(* Logix 5000 project; controller Oki_4_23 vendor 1 type 14 code 77 rev 20.12; software revision 20.01 *)

TASK MainTask (continuous, watchdog 500 ms) : MainProgram

MODULES
   Controller : vendor 1 type 14 code 77 (CompactLogixL32EController 0, rev 20.12)
      LocalENB : 1769-L32E Ethernet Port (CompactLogixL32Ethernet 1, rev 20.11)
      Local : CompactBus (CompactVirtualAdapter 3, rev 20.11)
         INPUT_1 : 1769-IQ16 (Compact 1, rev 1.1, Input RPI 20 ms)
         OUTPUT : 1769-OB16 (Compact 2, rev 2.1, Output RPI 20 ms)
END_MODULES

VAR_GLOBAL   (* controller tags *)
   GREEN : ALIAS FOR Local:2:O.Data.13;
   RED : ALIAS FOR Local:2:O.Data.15;
   START1 : ALIAS FOR Local:1:I.Data.1;
   START2 : ALIAS FOR Local:1:I.Data.2;
   START3 : ALIAS FOR Local:1:I.Data.3;
   START4 : ALIAS FOR Local:1:I.Data.4;
   STOP : ALIAS FOR Local:1:I.Data.5;
   TIMER1 : TIMER := (PRE := 5000);
   TIMER2 : TIMER := (PRE := 5000);
END_VAR

PROGRAM MainProgram   (* main routine MainRoutine *)

ROUTINE MainRoutine   (* ladder *)
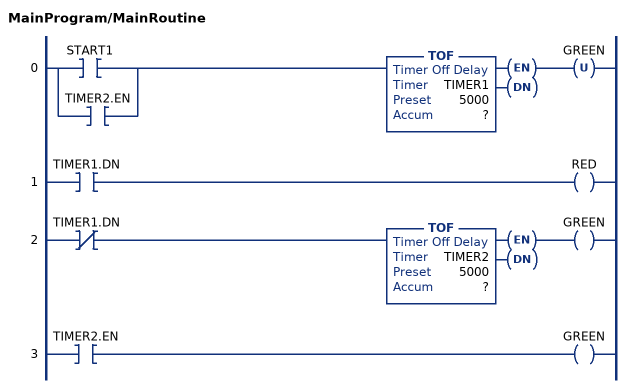
   0: [XIC(START1) ,XIC(TIMER2.EN) ]TOF(TIMER1,?,?)OTU(GREEN);
   1: XIC(TIMER1.DN)OTE(RED);
   2: XIO(TIMER1.DN)TOF(TIMER2,?,?)OTE(GREEN);
   3: XIC(TIMER2.EN)OTE(GREEN);
END_ROUTINE
END_PROGRAM
